PROGRAM SP3_3_Y132
VAR
	CompareOutput132_00: CMP_OC_DW;
	CompareOutput132_01: CMP_OC_DW;
	CompareOutput132_02: CMP_OC_DW;
	CompareOutput132_03: CMP_OC_DW;
	CompareOutput132_04: CMP_OC_DW;
	CompareOutput132_05: CMP_OC_DW;
	CompareOutput132_06: CMP_OC_DW;
	CompareOutput132_07: CMP_OC_DW;
	CompareOutput132_08: CMP_OC_DW;
	CompareOutput132_09: CMP_OC_DW;
	CompareOutput132_10: CMP_OC_DW;
	CompareOutput132_11: CMP_OC_DW;
	CompareOutput132_12: CMP_OC_DW;
	CompareOutput132_13: CMP_OC_DW;
	CompareOutput132_14: CMP_OC_DW;
	CompareOutput132_15: CMP_OC_DW;
END_VAR

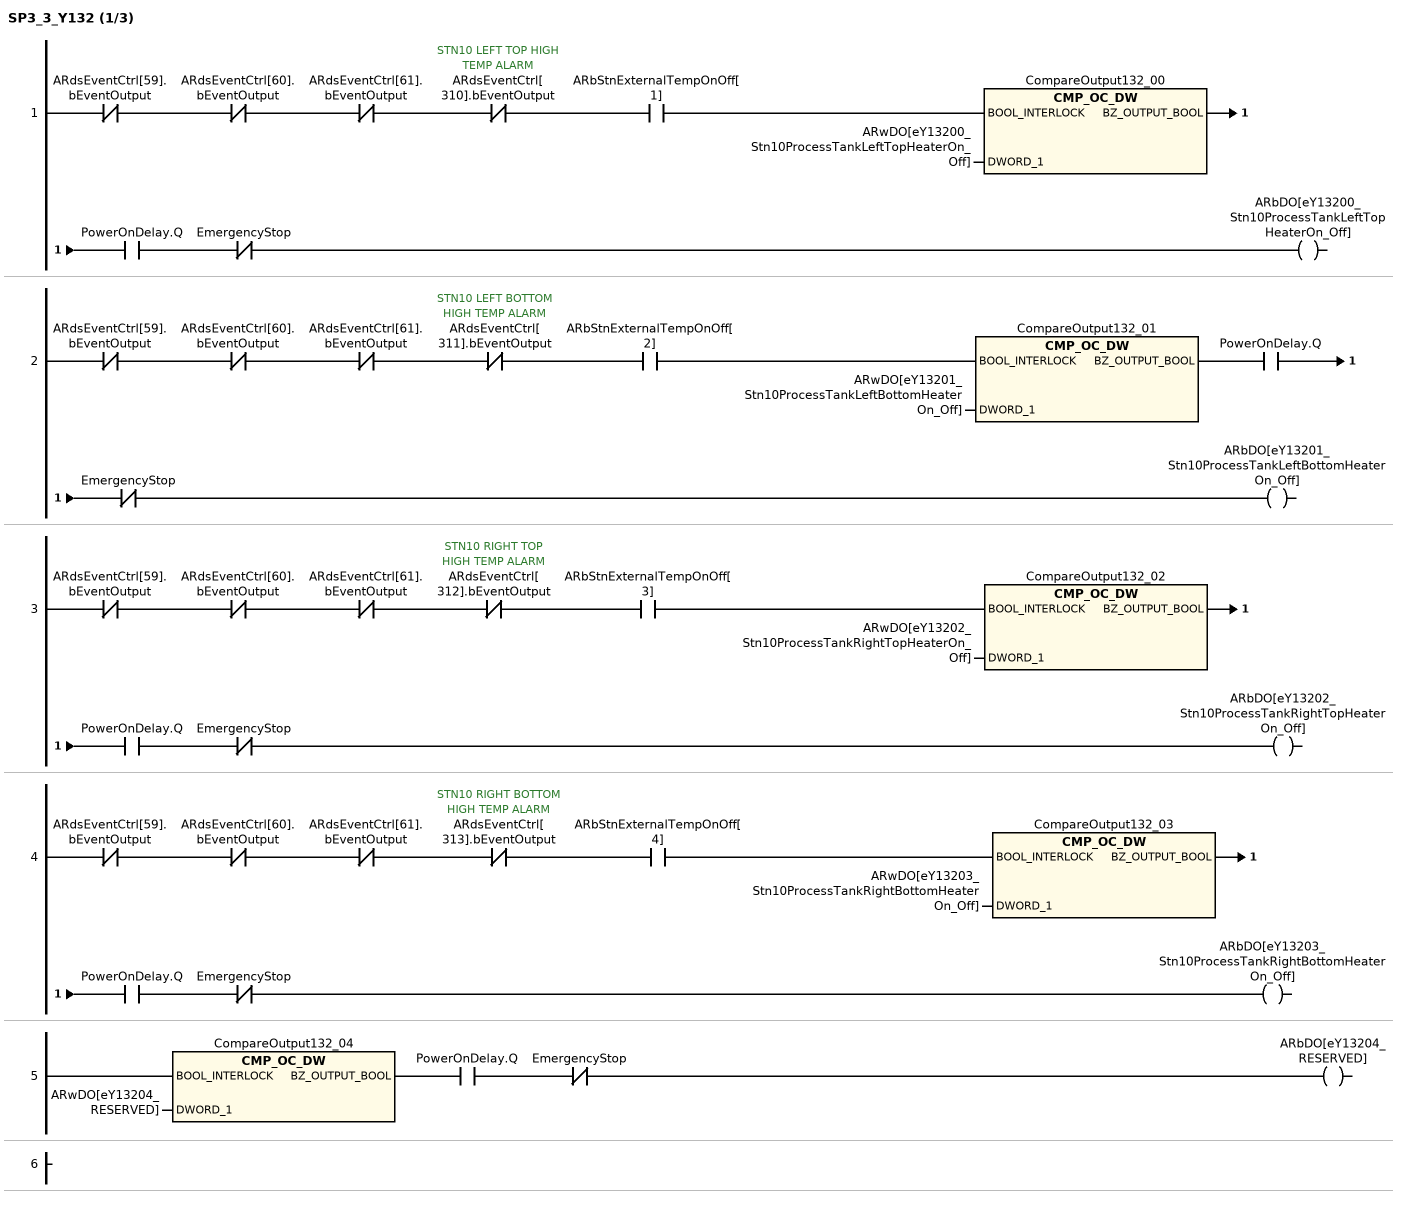
// NETWORK 1
//   ARdsEventCtrl[310].bEventOutput: STN10 LEFT TOP HIGH TEMP ALARM
CompareOutput132_00(BOOL_INTERLOCK := NOT ARdsEventCtrl[59].bEventOutput AND NOT ARdsEventCtrl[60].bEventOutput AND NOT ARdsEventCtrl[61].bEventOutput AND NOT ARdsEventCtrl[310].bEventOutput AND ARbStnExternalTempOnOff[1], DWORD_1 := ARwDO[eY13200_Stn10ProcessTankLeftTopHeaterOn_Off]); // CMP_OC_DW
ARbDO[eY13200_Stn10ProcessTankLeftTopHeaterOn_Off] := CompareOutput132_00.BZ_OUTPUT_BOOL AND PowerOnDelay.Q AND NOT EmergencyStop;

// NETWORK 2
//   ARdsEventCtrl[311].bEventOutput: STN10 LEFT BOTTOM HIGH TEMP ALARM
CompareOutput132_01(BOOL_INTERLOCK := NOT ARdsEventCtrl[59].bEventOutput AND NOT ARdsEventCtrl[60].bEventOutput AND NOT ARdsEventCtrl[61].bEventOutput AND NOT ARdsEventCtrl[311].bEventOutput AND ARbStnExternalTempOnOff[2], DWORD_1 := ARwDO[eY13201_Stn10ProcessTankLeftBottomHeaterOn_Off]); // CMP_OC_DW
ARbDO[eY13201_Stn10ProcessTankLeftBottomHeaterOn_Off] := CompareOutput132_01.BZ_OUTPUT_BOOL AND PowerOnDelay.Q AND NOT EmergencyStop;

// NETWORK 3
//   ARdsEventCtrl[312].bEventOutput: STN10 RIGHT TOP HIGH TEMP ALARM
CompareOutput132_02(BOOL_INTERLOCK := NOT ARdsEventCtrl[59].bEventOutput AND NOT ARdsEventCtrl[60].bEventOutput AND NOT ARdsEventCtrl[61].bEventOutput AND NOT ARdsEventCtrl[312].bEventOutput AND ARbStnExternalTempOnOff[3], DWORD_1 := ARwDO[eY13202_Stn10ProcessTankRightTopHeaterOn_Off]); // CMP_OC_DW
ARbDO[eY13202_Stn10ProcessTankRightTopHeaterOn_Off] := CompareOutput132_02.BZ_OUTPUT_BOOL AND PowerOnDelay.Q AND NOT EmergencyStop;

// NETWORK 4
//   ARdsEventCtrl[313].bEventOutput: STN10 RIGHT BOTTOM HIGH TEMP ALARM
CompareOutput132_03(BOOL_INTERLOCK := NOT ARdsEventCtrl[59].bEventOutput AND NOT ARdsEventCtrl[60].bEventOutput AND NOT ARdsEventCtrl[61].bEventOutput AND NOT ARdsEventCtrl[313].bEventOutput AND ARbStnExternalTempOnOff[4], DWORD_1 := ARwDO[eY13203_Stn10ProcessTankRightBottomHeaterOn_Off]); // CMP_OC_DW
ARbDO[eY13203_Stn10ProcessTankRightBottomHeaterOn_Off] := CompareOutput132_03.BZ_OUTPUT_BOOL AND PowerOnDelay.Q AND NOT EmergencyStop;

// NETWORK 5
CompareOutput132_04(BOOL_INTERLOCK := TRUE, DWORD_1 := ARwDO[eY13204_RESERVED]); // CMP_OC_DW
ARbDO[eY13204_RESERVED] := CompareOutput132_04.BZ_OUTPUT_BOOL AND PowerOnDelay.Q AND NOT EmergencyStop;

// NETWORK 6

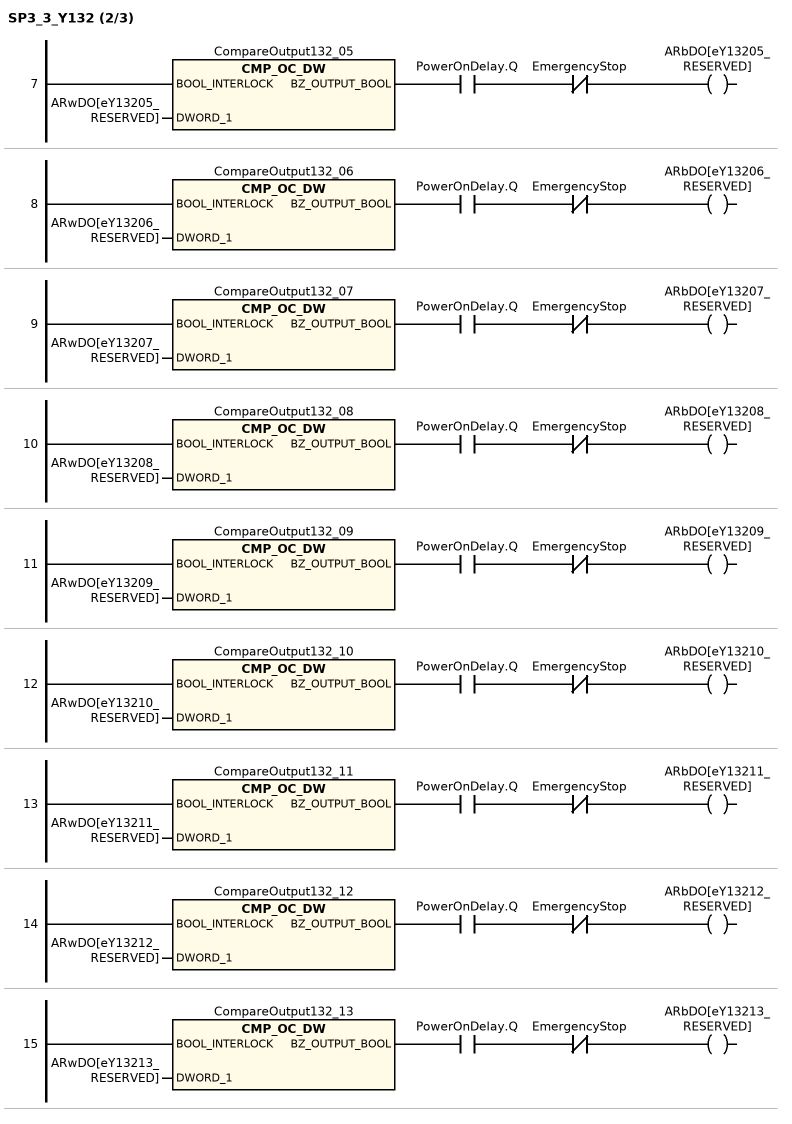
// NETWORK 7
CompareOutput132_05(BOOL_INTERLOCK := TRUE, DWORD_1 := ARwDO[eY13205_RESERVED]); // CMP_OC_DW
ARbDO[eY13205_RESERVED] := CompareOutput132_05.BZ_OUTPUT_BOOL AND PowerOnDelay.Q AND NOT EmergencyStop;

// NETWORK 8
CompareOutput132_06(BOOL_INTERLOCK := TRUE, DWORD_1 := ARwDO[eY13206_RESERVED]); // CMP_OC_DW
ARbDO[eY13206_RESERVED] := CompareOutput132_06.BZ_OUTPUT_BOOL AND PowerOnDelay.Q AND NOT EmergencyStop;

// NETWORK 9
CompareOutput132_07(BOOL_INTERLOCK := TRUE, DWORD_1 := ARwDO[eY13207_RESERVED]); // CMP_OC_DW
ARbDO[eY13207_RESERVED] := CompareOutput132_07.BZ_OUTPUT_BOOL AND PowerOnDelay.Q AND NOT EmergencyStop;

// NETWORK 10
CompareOutput132_08(BOOL_INTERLOCK := TRUE, DWORD_1 := ARwDO[eY13208_RESERVED]); // CMP_OC_DW
ARbDO[eY13208_RESERVED] := CompareOutput132_08.BZ_OUTPUT_BOOL AND PowerOnDelay.Q AND NOT EmergencyStop;

// NETWORK 11
CompareOutput132_09(BOOL_INTERLOCK := TRUE, DWORD_1 := ARwDO[eY13209_RESERVED]); // CMP_OC_DW
ARbDO[eY13209_RESERVED] := CompareOutput132_09.BZ_OUTPUT_BOOL AND PowerOnDelay.Q AND NOT EmergencyStop;

// NETWORK 12
CompareOutput132_10(BOOL_INTERLOCK := TRUE, DWORD_1 := ARwDO[eY13210_RESERVED]); // CMP_OC_DW
ARbDO[eY13210_RESERVED] := CompareOutput132_10.BZ_OUTPUT_BOOL AND PowerOnDelay.Q AND NOT EmergencyStop;

// NETWORK 13
CompareOutput132_11(BOOL_INTERLOCK := TRUE, DWORD_1 := ARwDO[eY13211_RESERVED]); // CMP_OC_DW
ARbDO[eY13211_RESERVED] := CompareOutput132_11.BZ_OUTPUT_BOOL AND PowerOnDelay.Q AND NOT EmergencyStop;

// NETWORK 14
CompareOutput132_12(BOOL_INTERLOCK := TRUE, DWORD_1 := ARwDO[eY13212_RESERVED]); // CMP_OC_DW
ARbDO[eY13212_RESERVED] := CompareOutput132_12.BZ_OUTPUT_BOOL AND PowerOnDelay.Q AND NOT EmergencyStop;

// NETWORK 15
CompareOutput132_13(BOOL_INTERLOCK := TRUE, DWORD_1 := ARwDO[eY13213_RESERVED]); // CMP_OC_DW
ARbDO[eY13213_RESERVED] := CompareOutput132_13.BZ_OUTPUT_BOOL AND PowerOnDelay.Q AND NOT EmergencyStop;

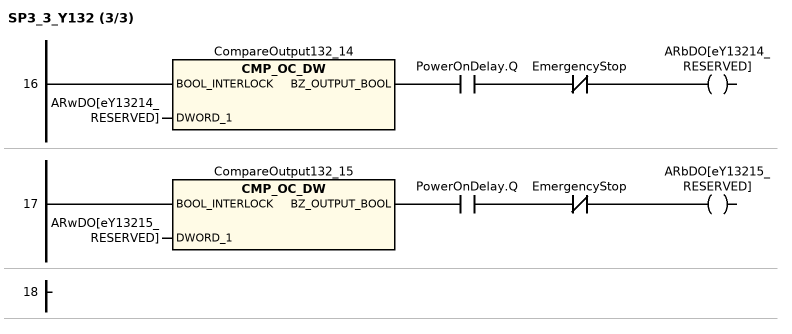
// NETWORK 16
CompareOutput132_14(BOOL_INTERLOCK := TRUE, DWORD_1 := ARwDO[eY13214_RESERVED]); // CMP_OC_DW
ARbDO[eY13214_RESERVED] := CompareOutput132_14.BZ_OUTPUT_BOOL AND PowerOnDelay.Q AND NOT EmergencyStop;

// NETWORK 17
CompareOutput132_15(BOOL_INTERLOCK := TRUE, DWORD_1 := ARwDO[eY13215_RESERVED]); // CMP_OC_DW
ARbDO[eY13215_RESERVED] := CompareOutput132_15.BZ_OUTPUT_BOOL AND PowerOnDelay.Q AND NOT EmergencyStop;

// NETWORK 18

END_PROGRAM

(* stored: Version 1.1.0.1, ProductVersion 3.1.4024.11
   POU SP3_3_Y132: Id {bf74678c-c47f-411e-a00c-5d2e06583df7}, SpecialFunc None *)
